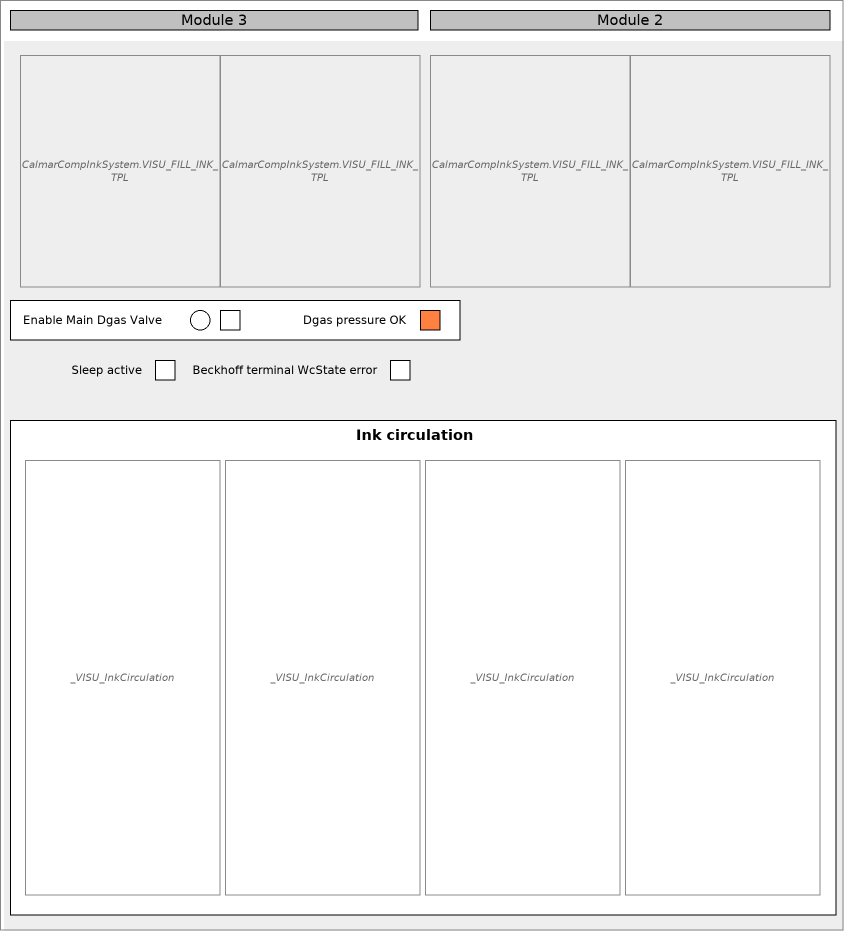
VISUALIZATION VISU_INK  // 844x931
    Rectangle (4,41 840x890)
    Rectangle (10,300 450x40)
    Ellipse (190,310 20x20), colour toggle: PRG_INK.bIDp_EnableMainDgasValve
        toggle PRG_INK.bIDp_EnableMainDgasValve
    Rectangle (20,310 160x20), "Enable Main Dgas Valve"
    RoundedRectangle (220,310 20x20), colour toggle: PRG_INK.bODp_EnableMainDgasValve
    Rectangle (300,310 110x20), "Dgas pressure OK"
    RoundedRectangle (420,310 20x20), colour toggle: PRG_INK.bODp_DgasPressOK
    RoundedRectangle (155,360 20x20), colour toggle: PRG_MACHINE.sO_SystemCmd.bSleep
    Rectangle (70,360 75x20), "Sleep active"
    RoundedRectangle (390,360 20x20), colour toggle: PRG_INK.bI_InkLevel1WcState
    Rectangle (190,360 190x20), "Beckhoff terminal WcState error"
    Frame (20,55 200x232)
        shows CalmarCompInkSystem.VISU_FILL_INK_TPL(m_InkDegasExisting := CONFIGURATION.bCIk_INK_DEGASSING_EXISTING, m_ModId_StAdsHeadertank := PRG_INK.sAdsIkHeaderTank[4], m_ModId_StAdsInkPump := PRG_INK.sAdsIkInkPump[4], m_ModId_FbInkSupply := PRG_INK.fb_FillInkVarnish[4], m_ModId_StInkDefinition := PRG_INK.sL_InkTable[4])
    Frame (220,55 200x232)
        shows CalmarCompInkSystem.VISU_FILL_INK_TPL(m_InkDegasExisting := CONFIGURATION.bCIk_INK_DEGASSING_EXISTING, m_ModId_StAdsHeadertank := PRG_INK.sAdsIkHeaderTank[3], m_ModId_StAdsInkPump := PRG_INK.sAdsIkInkPump[3], m_ModId_FbInkSupply := PRG_INK.fb_FillInkVarnish[3], m_ModId_StInkDefinition := PRG_INK.sL_InkTable[3])
    Frame (430,55 200x232)
        shows CalmarCompInkSystem.VISU_FILL_INK_TPL(m_InkDegasExisting := CONFIGURATION.bCIk_INK_DEGASSING_EXISTING, m_ModId_StAdsHeadertank := PRG_INK.sAdsIkHeaderTank[2], m_ModId_StAdsInkPump := PRG_INK.sAdsIkInkPump[2], m_ModId_FbInkSupply := PRG_INK.fb_FillInkVarnish[2], m_ModId_StInkDefinition := PRG_INK.sL_InkTable[2])
    Frame (630,55 200x232)
        shows CalmarCompInkSystem.VISU_FILL_INK_TPL(m_InkDegasExisting := CONFIGURATION.bCIk_INK_DEGASSING_EXISTING, m_ModId_StAdsHeadertank := PRG_INK.sAdsIkHeaderTank[1], m_ModId_StAdsInkPump := PRG_INK.sAdsIkInkPump[1], m_ModId_FbInkSupply := PRG_INK.fb_FillInkVarnish[1], m_ModId_StInkDefinition := PRG_INK.sL_InkTable[1])
    Rectangle (10,420 826x495)
    Rectangle (335,425 160x20), "Ink circulation"
    Frame (625,460 195x435)
        shows _VISU_InkCirculation(m_Inst_Fb := PRG_INK.fb_CirculationInk[1])
    Frame (425,460 195x435)
        shows _VISU_InkCirculation(m_Inst_Fb := PRG_INK.fb_CirculationInk[2])
    Frame (225,460 195x435)
        shows _VISU_InkCirculation(m_Inst_Fb := PRG_INK.fb_CirculationInk[3])
    Frame (25,460 195x435)
        shows _VISU_InkCirculation(m_Inst_Fb := PRG_INK.fb_CirculationInk[4])
    Rectangle (10,10 408x20), "Module 3"
    Rectangle (430,10 400x20), "Module 2"
END_VISUALIZATION

(* stored: Version 1.1.0.1, ProductVersion 3.1.4024.9
   Visu VISU_INK: Id {1362828b-338e-4fd7-bdf1-2745a1174815} *)
